(* CODESYS project RepPublic

Project tree, tasks and I/O mapping:
  Device : CODESYS Control Win V3 x64, 3S - Smart Software Solutions GmbH, version 3.5.18.20
    application Application
      libraries: Standard, 3.5.18.0 (System)
      task MainTask (cyclic, interval t#20ms, priority 1) calls PLC_PRG
      task TaskHugo (cyclic, interval t#20ms, priority 1) calls _Hugo
      task TaskHugo (cyclic, interval t#20ms, priority 1) calls _Hugo
      HUGO/
        program _Hugo [ST]
      HUGO/
        program _Hugo [ST]
      program PLC_PRG [ST]
*)

// Device/Application/PLC_PRG
PROGRAM PLC_PRG
VAR
	Hugo: INT;
END_VAR

Hugo := Hugo +1;

END_PROGRAM

// Device/Application/HUGO/_Hugo
//. automatic generated Hugo PRG, DF, CODESYS Academy
PROGRAM _Hugo
VAR
	Hugo : INT;
END_VAR

Hugo := Hugo +1;

END_PROGRAM

// Device/Application/HUGO/_Hugo
//.{attribute 'analysis' := '-*'}
//. automatic generated Hugo PRG, DF, CODESYS Academy
PROGRAM _Hugo
VAR
	Hugo : INT;
END_VAR

Hugo := Hugo +1;

END_PROGRAM
